{attribute 'qualified_only'}
{attribute 'strict'}
TYPE e_Displacement :
(
	eNoDisplacement := 1<<0, eMoveStraight := 1<<1, eBezierCurve := 1<<2, ePathfinding := 1<<3
);
END_TYPE

(* stored: Version 1.1.0.1, ProductVersion 3.1.4022.18
   DUT e_Displacement: Id {f6f03fbe-f8e3-4f70-b79d-864318635ee6} *)
